PROGRAM PRG_MachineConfigure
VAR
END_VAR

IF (NOT GVL_SystemVariable.bMachineInitDone) THEN

//	GVL_SystemConfigure.fbMachineConfigure.AddConfiguration (fbConfigure := GVL_MachineVariable.fbMachineConfiguration);
//	GVL_SystemConfigure.fbHMIConfigure.AddConfiguration (fbConfigure := GVL_MachineVariable.fbHMIConfiguration);
	GVL_SystemVariable.bMachineInitDone		:= TRUE;
END_IF

END_PROGRAM

(* stored: Version 1.1.0.1, ProductVersion 3.1.4024.15
   POU PRG_MachineConfigure: Id {3a3f2f0a-85ff-4c45-9b85-749efe215256}, SpecialFunc None *)
